(* PLC project Unnamed, Unknown Unnamed 1 *)
(* stored: creationDateTime 2022-10-30T21:25:48, modificationDateTime 2022-10-31T09:14:30 *)

PROGRAM TC005
  VAR_INPUT
    i1 : BOOL;
    i2 : BOOL := FALSE;
  END_VAR
  VAR_OUTPUT
    o1 : BOOL := FALSE;
    o2 : BOOL := FALSE;
  END_VAR
  VAR
    i3 : TIME := T#5s;
    o4 : BOOL;
    TON0 : TON;
  END_VAR
  VAR  (* added by the conversion: wires and edge detectors of the diagram *)
    _AND1_OUT : BOOL;
    _XOR3_OUT : BOOL;
  END_VAR

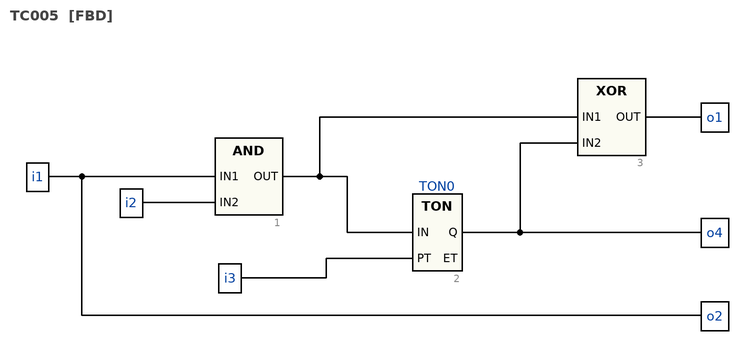
(* FBD diagram, written out as Structured Text *)
_AND1_OUT := i1 AND i2;
TON0(IN := _AND1_OUT, PT := i3);
_XOR3_OUT := _AND1_OUT XOR TON0.Q;
o1 := _XOR3_OUT;
o4 := TON0.Q;
o2 := i1;
END_PROGRAM

CONFIGURATION config
  RESOURCE resource1 ON PLC
  END_RESOURCE
END_CONFIGURATION
